TYPE inserterUnLoadIO :
STRUCT
	
	// Входове
	x_Grip_open				: BOOL;           // Грипера е отворен - сензор на цилиндър
    x_Grip_close            : BOOL;           // Грипера е затворен - сензор на цилиндър
	x_Insert_up             : BOOL;           // Инсъртъра е вдигнат - сензор на цилиндър
	x_Insert_down           : BOOL;           // Инсъртъра е свален	- сензор на цилиндър
	x_Nest                  : BOOL;           // Лазърен сензор - детектва имали продукт в гнездото под инсъртъра
	
	// Изходи
	y_Grip_open				: BOOL;           // Грипера е отворен -  цилиндър
    y_Grip_close            : BOOL;           // Грипера е затворен -  цилиндър
	y_Insert_up             : BOOL;           // Инсъртъра е вдигнат - цилиндър
	y_Insert_down           : BOOL;           // Инсъртъра е свален	-  цилиндър

END_STRUCT
END_TYPE

(* stored: Version 1.1.0.1, ProductVersion 3.1.4024.3
   DUT inserterUnLoadIO: Id {61977c55-1c72-4686-b58c-a73dd455e8e1} *)
